(* PLC project SansNom, Inconnu SansNom 1 *)
(* stored: creationDateTime 2024-11-06T09:39:17, modificationDateTime 2024-11-06T11:56:14 *)

PROGRAM program0
  VAR
    LocalVar0 : DINT;
  END_VAR

(* LD diagram, written out as Structured Text *)
END_PROGRAM

CONFIGURATION Config0
  RESOURCE Res0 ON PLC
    VAR_GLOBAL
      LocalVar0 : DINT;
      LocalVar3 : DINT;
      LocalVar1 : DINT;
      LocalVar2 : DINT;
    END_VAR
    TASK task0(INTERVAL := T#20ms, PRIORITY := 0);
    PROGRAM instance0 WITH task0 : program0;
    PROGRAM instance1 WITH task0 : program0;
  END_RESOURCE
  RESOURCE resource0 ON PLC
  END_RESOURCE
END_CONFIGURATION
